FUNCTION F_PB_GetZoneITC : ST_ITC_Zone
VAR_INPUT
		eFunctionNumber		: E_FunctionNumber; // Function number
		ZoneNumber			: INT := 1;
END_VAR
VAR
END_VAR

// Check if function number is validas
IF eFunctionNumber > E_FunctionNumber.F_BEGIN_FUNCTION AND
   eFunctionNumber < E_FunctionNumber.F_END_FUNCTION THEN
  
	// Check reference is valid
	IF __ISVALIDREF(FunctionRegistry[eFunctionNumber].rFunctionInterface) THEN
   		// Return function interlock
   		F_PB_GetZoneITC := FunctionRegistry[eFunctionNumber].rFunction.ITC.ZoneITC[ZoneNumber];
	END_IF
END_IF

END_FUNCTION

(* stored: Version 1.1.0.1, ProductVersion 3.1.4022.12
   POU F_PB_GetZoneITC: Id {617e4b42-8cf0-4c08-ac53-f2cbbee96776}, SpecialFunc None *)
